// TIA Portal project "Washing Machine" (V16)

(* hardware
DEVICE "S7-1200 station_1"  S7-1200 Station
   slot 0: "Rack_0"  S7-1200 Rack  Rack  V1.0
   slot 1: "PLC_1"  CPU 1212C AC/DC/Rly  6ES7 212-1BE40-0XB0  V4.0
*)

// ===== PLC "PLC_1"  CPU 1212C AC/DC/Rly =====

VAR_GLOBAL   // PLC tag table "Default tag table"
   "start" AT %I0.2 : Bool;
   "K1" AT %Q0.0 : Bool;
   "stop1" AT %I0.4 : Bool;
   "k2" AT %Q0.1 : Bool;
   "STOP" AT %I0.3 : Bool;
   "T1 tag" AT %M0.0 : Bool;
   "T2 tag" AT %M0.1 : Bool;
   "X" AT %M0.2 : Bool;
   "T3 tag" AT %M0.3 : Bool;
   "T4 tag" AT %M0.4 : Bool;
   "Tag_1" AT %M0.5 : Bool;
   "Tag_2" AT %M0.6 : Bool;
END_VAR

// folder: System blocks/Program resources

DATA_BLOCK "T1"   // DB2
{ S7_Optimized_Access := 'TRUE' }
AUTHOR : Simatic
FAMILY : IEC
NAME : IEC_TMR
VERSION : 1.0
// stored: InstanceOfName IEC_TIMER
"IEC_TIMER"
BEGIN
END_DATA_BLOCK

DATA_BLOCK "T2"   // DB3
{ S7_Optimized_Access := 'TRUE' }
AUTHOR : Simatic
FAMILY : IEC
NAME : IEC_TMR
VERSION : 1.0
// stored: InstanceOfName IEC_TIMER
"IEC_TIMER"
BEGIN
END_DATA_BLOCK

DATA_BLOCK "T3"   // DB4
{ S7_Optimized_Access := 'TRUE' }
AUTHOR : Simatic
FAMILY : IEC
NAME : IEC_TMR
VERSION : 1.0
// stored: InstanceOfName IEC_TIMER
"IEC_TIMER"
BEGIN
END_DATA_BLOCK

DATA_BLOCK "T4"   // DB5
{ S7_Optimized_Access := 'TRUE' }
AUTHOR : Simatic
FAMILY : IEC
NAME : IEC_TMR
VERSION : 1.0
// stored: InstanceOfName IEC_TIMER
"IEC_TIMER"
BEGIN
END_DATA_BLOCK

// folder: (top level)

ORGANIZATION_BLOCK "Main"   // OB1, LAD, ProgramCycle
TITLE = "Main Program Sweep (Cycle)"
{ S7_Optimized_Access := 'TRUE' }
VERSION : 0.1
   VAR_INPUT
      Initial_Call : Bool;   // Initial call of this OB
      Remanence : Bool;   // =True, if remanent data are available
   END_VAR
BEGIN

REGION Network 1: start
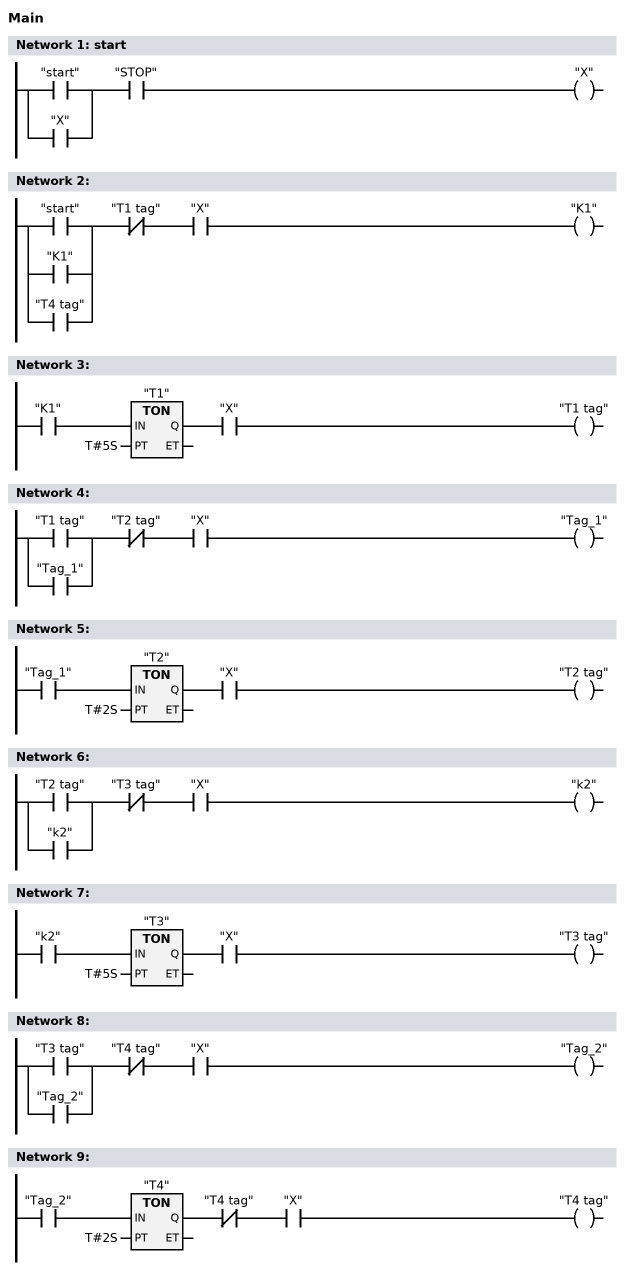
   RUNG wire#powerrail
      Contact( "start" )
      wire#w1
      Contact( "STOP" )
      Coil( "X" )
   END_RUNG
   RUNG wire#powerrail
      Contact( "X" )
   END_RUNG wire#w1
   // the same network as SCL:
   "X" := ("start" OR "X") AND "STOP";
END_REGION

REGION Network 2
   RUNG wire#powerrail
      Contact( "start" )
      wire#w1
      I_Contact( "T1 tag" )
      Contact( "X" )
      Coil( "K1" )
   END_RUNG
   RUNG wire#powerrail
      Contact( "K1" )
   END_RUNG wire#w1
   RUNG wire#powerrail
      Contact( "T4 tag" )
   END_RUNG wire#w1
   // the same network as SCL:
   "K1" := ("start" OR "K1" OR "T4 tag") AND NOT "T1 tag" AND "X";
END_REGION

REGION Network 3
   "T1".TON(IN := "K1", PT := T#5S);
   "T1 tag" := "T1".Q AND "X";
END_REGION

REGION Network 4
   RUNG wire#powerrail
      Contact( "T1 tag" )
      wire#w1
      I_Contact( "T2 tag" )
      Contact( "X" )
      Coil( "Tag_1" )
   END_RUNG
   RUNG wire#powerrail
      Contact( "Tag_1" )
   END_RUNG wire#w1
   // the same network as SCL:
   "Tag_1" := ("T1 tag" OR "Tag_1") AND NOT "T2 tag" AND "X";
END_REGION

REGION Network 5
   "T2".TON(IN := "Tag_1", PT := T#2S);
   "T2 tag" := "T2".Q AND "X";
END_REGION

REGION Network 6
   RUNG wire#powerrail
      Contact( "T2 tag" )
      wire#w1
      I_Contact( "T3 tag" )
      Contact( "X" )
      Coil( "k2" )
   END_RUNG
   RUNG wire#powerrail
      Contact( "k2" )
   END_RUNG wire#w1
   // the same network as SCL:
   "k2" := ("T2 tag" OR "k2") AND NOT "T3 tag" AND "X";
END_REGION

REGION Network 7
   "T3".TON(IN := "k2", PT := T#5S);
   "T3 tag" := "T3".Q AND "X";
END_REGION

REGION Network 8
   RUNG wire#powerrail
      Contact( "T3 tag" )
      wire#w1
      I_Contact( "T4 tag" )
      Contact( "X" )
      Coil( "Tag_2" )
   END_RUNG
   RUNG wire#powerrail
      Contact( "Tag_2" )
   END_RUNG wire#w1
   // the same network as SCL:
   "Tag_2" := ("T3 tag" OR "Tag_2") AND NOT "T4 tag" AND "X";
END_REGION

REGION Network 9
   "T4".TON(IN := "Tag_2", PT := T#2S);
   "T4 tag" := "T4".Q AND NOT "T4 tag" AND "X";
END_REGION
END_ORGANIZATION_BLOCK